FUNCTION_BLOCK List_Person_Test EXTENDS TcUnit.FB_TestSuite

AddAndGet();
AddAndGetShouldBeByReference();
GetCapacity();
GetCount();
Clear();
RemoveAt();
RemoveRange();
Contains();
Exists();
Find();
FindAll();
FindIndex();
FindLast();
FindLastIndex();
Foreach();

METHOD AddAndGet
VAR
    list_Person_ : List_Person_;
    expectedPerson : Person;
    expectedAge : INT := 10;
    expectedIndex : INT := 0;
    actualPtPerson : POINTER TO Person;
    actualAge : INT;
    actualIndex : INT;
END_VAR
TEST('AddAndGetPersonShouldPass');

//Assign
expectedPerson.SetAge(expectedAge);

//Act
actualIndex := list_Person_.AddItem(expectedPerson);
actualPtPerson := list_Person_.GetItem(actualIndex);
actualAge := actualPtPerson^.GetAge();

//Assert
AssertEquals(expectedIndex, actualIndex,'');
AssertEquals(expectedAge, actualAge,'');
AssertTrue(actualPtPerson^.Equals(expectedPerson),'');


TEST_FINISHED();
END_METHOD

METHOD AddAndGetShouldBeByReference
VAR
    list_Person_ : List_Person_;
    expectedPerson : Person;
    expectedAge : INT := 10;
    actualPtPerson : POINTER TO Person;
    actualAge : INT;
END_VAR
TEST('AddAndGetShouldBeByReference');

//Assign

//Act
list_Person_.AddItem(expectedPerson);
actualPtPerson := list_Person_.GetItem(0);
expectedPerson.SetAge(expectedAge);
actualAge := actualPtPerson^.GetAge();

//Assert
AssertEquals(expectedAge, actualAge,'');


TEST_FINISHED();
END_METHOD

METHOD Clear
VAR
    list_Person_ : List_Person_;
    person : Person;
    expectedCount : INT := 1;
    actualCount : INT;
END_VAR
TEST('ClearShouldPass');

//Assign
list_Person_.AddItem(person);

//Act
actualCount := list_Person_.GetCount();

//Assert
AssertEquals(expectedCount, actualCount,'Get count after adding a person');

//Act
list_Person_.Clear();
actualCount := list_Person_.GetCount();

//Assert
expectedCount := 0;
AssertEquals(expectedCount, actualCount,'Get count after clearing the list');


TEST_FINISHED();
END_METHOD

METHOD Contains
VAR
    list_Person_ : List_Person_;
    personA : Person;
    personB : Person;
    personC : Person;
    personD : Person;
    personE : Person;
    personF : Person;
    personG : Person;
    actual : BOOL;
    expected : BOOL := TRUE;
END_VAR
TEST('ContainsShouldPass');

//Assign
personA.SetAge(10);
personB.SetAge(11);
personC.SetAge(12);
personD.SetAge(13);
personE.SetAge(14);
personF.SetAge(15);
personG.SetAge(16);
personA.SetName('A');
personB.SetName('B');
personC.SetName('C');
personD.SetName('D');
personE.SetName('E');
personF.SetName('F');
personG.SetName('G');
list_Person_.AddItem(personA);
list_Person_.AddItem(personB);
list_Person_.AddItem(personC);
list_Person_.AddItem(personD);
list_Person_.AddItem(personE);
list_Person_.AddItem(personF);

//Act
actual := list_Person_.Contains(personC);

//Assert
AssertEquals(expected, actual,'Looking for personC');

//Act
actual := list_Person_.Contains(personG);

//Assert
expected := FALSE;
AssertEquals(expected, actual,'Looking for personG');


TEST_FINISHED();
END_METHOD

METHOD Exists
VAR
    list_Person_ : List_Person_;
    personA : Person;
    personB : Person;
    personC : Person;
    personD : Person;
    personE : Person;
    personF : Person;
    personG : Person;
    predicate_Person_ : Predicate_Person_;
    actual : BOOL;
    expected : BOOL := TRUE;
END_VAR
TEST('ExistsShouldPass');

//Assign
personA.SetAge(10);
personB.SetAge(11);
personC.SetAge(12);
personD.SetAge(13);
personE.SetAge(14);
personF.SetAge(15);
personG.SetAge(16);
personA.SetName('A');
personB.SetName('B');
personC.SetName('C');
personD.SetName('D');
personE.SetName('E');
personF.SetName('F');
personG.SetName('G');
list_Person_.AddItem(personA);
list_Person_.AddItem(personB);
list_Person_.AddItem(personC);
list_Person_.AddItem(personD);
list_Person_.AddItem(personE);
list_Person_.AddItem(personF);

//Act
actual := list_Person_.Exists(predicate_Person_, 2);

//Assert
AssertEquals(expected, actual,'Looking for a person with name C');

//Act
actual := list_Person_.Exists(predicate_Person_, 3);

//Assert
expected := FALSE;
AssertEquals(expected, actual,'Looking for a person with name G');


TEST_FINISHED();
END_METHOD

METHOD Find
VAR
    list_Person_ : List_Person_;
    personA : Person;
    personB : Person;
    personC : Person;
    personD : Person;
    personE : Person;
    personF : Person;
    personG : Person;
    predicate_Person_ : Predicate_Person_;
    actualPtPerson : POINTER TO Person;
    nullPtPerson : POINTER TO person := 0;
END_VAR
TEST('FindShouldPass');

//Assign
personA.SetAge(10);
personB.SetAge(11);
personC.SetAge(12);
personD.SetAge(13);
personE.SetAge(14);
personF.SetAge(15);
personG.SetAge(16);
personA.SetName('A');
personB.SetName('B');
personC.SetName('C');
personD.SetName('D');
personE.SetName('E');
personF.SetName('F');
personG.SetName('G');
list_Person_.AddItem(personA);
list_Person_.AddItem(personB);
list_Person_.AddItem(personC);
list_Person_.AddItem(personD);
list_Person_.AddItem(personE);
list_Person_.AddItem(personF);

//Act
actualPtPerson := list_Person_.Find(predicate_Person_, 2);

//Assert
AssertTrue(actualPtPerson^.Equals(personC),'Get person with name C');

//Act
actualPtPerson := list_Person_.Find(predicate_Person_, 3);

//Assert
AssertEquals(nullPtPerson, actualPtPerson,'Get Zero when looking for person with name G');


TEST_FINISHED();
END_METHOD

METHOD FindAll
VAR
    list_Person_ : List_Person_;
    personA : Person;
    personB : Person;
    personC : Person;
    personD : Person;
    personE : Person;
    personF : Person;
    personG : Person;
    predicate_Person_ : Predicate_Person_;
    actualList_Person_ : list_Person_;
    actualCount : INT;
    expectedCount : INT := 3;
    actualPtPerson0 : POINTER TO Person;
    actualPtPerson1 : POINTER TO Person;
    actualPtPerson2 : POINTER TO Person;
END_VAR
TEST('FindAllShouldPass');

//Assign
personA.SetAge(10);
personB.SetAge(11);
personC.SetAge(12);
personD.SetAge(13);
personE.SetAge(14);
personF.SetAge(15);
personG.SetAge(16);
list_Person_.AddItem(personA);
list_Person_.AddItem(personB);
list_Person_.AddItem(personC);
list_Person_.AddItem(personD);
list_Person_.AddItem(personE);
list_Person_.AddItem(personF);

//Act
actualList_Person_ := list_Person_.FindAll(predicate_Person_, 1); //Get people younger than 13
actualCount := actualList_Person_.GetCount();
actualPtPerson0 := actualList_Person_.GetItem(0);
actualPtPerson1 := actualList_Person_.GetItem(1);
actualPtPerson2 := actualList_Person_.GetItem(2);

//Assert
AssertEquals(expectedCount, actualCount, 'Check new list count');
AssertTrue(actualPtPerson0^.Equals(personA),'First element should personA');
AssertTrue(actualPtPerson1^.Equals(personB),'First element should personB');
AssertTrue(actualPtPerson2^.Equals(personC),'First element should personC');

TEST_FINISHED();
END_METHOD

METHOD FindIndex
VAR
    list_Person_ : List_Person_;
    personA : Person;
    personB : Person;
    personC : Person;
    personD : Person;
    personE : Person;
    personF : Person;
    personG : Person;
    predicate_Person_ : Predicate_Person_;
    actualIndex : INT;
    expectedIndex : INT := 2;
END_VAR
TEST('FindIndexShouldPass');

//Assign
personA.SetAge(10);
personB.SetAge(11);
personC.SetAge(12);
personD.SetAge(13);
personE.SetAge(14);
personF.SetAge(15);
personG.SetAge(16);
personA.SetName('A');
personB.SetName('B');
personC.SetName('C');
personD.SetName('D');
personE.SetName('E');
personF.SetName('F');
personG.SetName('G');
list_Person_.AddItem(personA);
list_Person_.AddItem(personB);
list_Person_.AddItem(personC);
list_Person_.AddItem(personD);
list_Person_.AddItem(personE);
list_Person_.AddItem(personF);

//Act
actualIndex := list_Person_.FindIndex(predicate_Person_, 2);

//Assert
AssertEquals(expectedIndex, actualIndex, 'find person with name C index');

//Act
actualIndex := list_Person_.FindIndex(predicate_Person_, 3);

//Assert
expectedIndex := -1;
AssertEquals(expectedIndex, actualIndex, 'Find person with name G index');


TEST_FINISHED();
END_METHOD

METHOD FindLast
VAR
    list_Person_ : List_Person_;
    personA : Person;
    personB : Person;
    personC : Person;
    personC2 : Person;
    personD : Person;
    personE : Person;
    personF : Person;
    personG : Person;
    predicate_Person_ : Predicate_Person_;
    actualPtPerson : POINTER TO Person;
    nullPtPerson : POINTER TO person := 0;
END_VAR
TEST('FindLastShouldPass');

//Assign
personA.SetAge(10);
personB.SetAge(11);
personC.SetAge(12);
personC2.SetAge(22);
personD.SetAge(13);
personE.SetAge(14);
personF.SetAge(15);
personG.SetAge(16);
personA.SetName('A');
personB.SetName('B');
personC.SetName('C');
personC2.SetName('C');
personD.SetName('D');
personE.SetName('E');
personF.SetName('F');
personG.SetName('G');
list_Person_.AddItem(personA);
list_Person_.AddItem(personB);
list_Person_.AddItem(personC);
list_Person_.AddItem(personD);
list_Person_.AddItem(personE);
list_Person_.AddItem(personC2); //Duplicated C
list_Person_.AddItem(personF);

//Act
actualPtPerson := list_Person_.FindLast(predicate_Person_, 2);

//Assert
AssertFalse(actualPtPerson^.Equals(personC),'Not the last person with name C');
AssertTrue(actualPtPerson^.Equals(personC2),'Be the last person with name C');

//Act
actualPtPerson := list_Person_.Find(predicate_Person_, 3);

//Assert
AssertEquals(nullPtPerson, actualPtPerson,'Get Zero when looking for person with name G');


TEST_FINISHED();
END_METHOD

METHOD FindLastIndex
VAR
    list_Person_ : List_Person_;
    personA : Person;
    personB : Person;
    personC : Person;
    personC2 : Person;
    personD : Person;
    personE : Person;
    personF : Person;
    personG : Person;
    predicate_Person_ : Predicate_Person_;
    actualIndex : INT;
    expectedIndex : INT := 5;
END_VAR
TEST('FindLastIndexShouldPass');

//Assign
personA.SetAge(10);
personB.SetAge(11);
personC.SetAge(12);
personC.SetAge(22);
personD.SetAge(13);
personE.SetAge(14);
personF.SetAge(15);
personG.SetAge(16);
personA.SetName('A');
personB.SetName('B');
personC.SetName('C');
personC2.SetName('C');
personD.SetName('D');
personE.SetName('E');
personF.SetName('F');
personG.SetName('G');
list_Person_.AddItem(personA);
list_Person_.AddItem(personB);
list_Person_.AddItem(personC);
list_Person_.AddItem(personD);
list_Person_.AddItem(personE);
list_Person_.AddItem(personC2);
list_Person_.AddItem(personF);

//Act
actualIndex := list_Person_.FindLastIndex(predicate_Person_, 2);

//Assert
AssertEquals(expectedIndex, actualIndex, 'Find last person with name C index');

//Act
actualIndex := list_Person_.FindLastIndex(predicate_Person_, 3);

//Assert
expectedIndex := -1;
AssertEquals(expectedIndex, actualIndex, 'Find person with name G index');


TEST_FINISHED();
END_METHOD

METHOD Foreach
VAR
    list_Person_ : List_Person_;
    personA : Person;
    personB : Person;
    personC : Person;
    personD : Person;
    personE : Person;
    personF : Person;
    personG : Person;
    action_Person_ : Action_Person_;
    actualPtPersonArray : ARRAY[0..3] OF POINTER TO Person;
    j : INT;
    expectedName : STRING := 'John';
END_VAR
TEST('ForeachShouldPass');

//Assign
personA.SetAge(10);
personB.SetAge(11);
personC.SetAge(12);
personD.SetAge(13);
personE.SetAge(14);
personF.SetAge(15);
personG.SetAge(16);
personA.SetName('A');
personB.SetName('B');
personC.SetName('C');
personD.SetName('D');
personE.SetName('E');
personF.SetName('F');
personG.SetName('G');
list_Person_.AddItem(personA);
list_Person_.AddItem(personB);
list_Person_.AddItem(personC);
list_Person_.AddItem(personD);

//Act
list_Person_.Foreach(action_Person_, 2);
FOR j:=0 TO 3 DO
    actualPtPersonArray[j] := list_Person_.GetItem(j);
END_FOR

//Assert
AssertEquals_STRING(expectedName, actualPtPersonArray[0]^.GetName(),'element 0 shuold be named John');
AssertEquals_STRING(expectedName, actualPtPersonArray[1]^.GetName(),'element 0 shuold be named John');
AssertEquals_STRING(expectedName, actualPtPersonArray[2]^.GetName(),'element 0 shuold be named John');
AssertEquals_STRING(expectedName, actualPtPersonArray[3]^.GetName(),'element 0 shuold be named John');


TEST_FINISHED();
END_METHOD

METHOD GetCapacity
VAR
    list_Person_ : List_Person_;
    person : Person;
    expectedCapacity : INT := GVL.LIST_UPPER_BOUND + 1;
    actualCapacity : INT;
END_VAR
TEST('GetCapacityShouldPass');

//Act
actualCapacity := list_Person_.GetCapacity();

//Assert1
AssertEquals_INT(expectedCapacity, actualCapacity,'Get capacity at the begining');


//Assign
list_Person_.AddItem(person);

//Act
actualCapacity := list_Person_.GetCapacity();

//Assert2
AssertEquals(expectedCapacity, actualCapacity,'Get capacity after adding a person');


TEST_FINISHED();
END_METHOD

METHOD GetCount
VAR
    list_Person_ : List_Person_;
    person : Person;
    expectedCount : INT := 0;
    actualCount : INT;
    actualPtPerson : POINTER TO Person;
END_VAR
TEST('GetCountShouldPass');

//Act
actualCount := list_Person_.GetCount();

//Assert
AssertEquals_INT(expectedCount, actualCount,'Get count at the begining');


//Assign
list_Person_.AddItem(person);

//Act
actualCount := list_Person_.GetCount();

//Assert
expectedCount := 1;
AssertEquals(expectedCount, actualCount,'Get count after adding a person');


TEST_FINISHED();
END_METHOD

METHOD RemoveAt
VAR
    list_Person_ : List_Person_;
    person : Person;
    expectedPtPerson : POINTER TO Person := 0;
    expectedCount : INT := 0;
    actualPtPerson : POINTER TO Person;
    actualCount : INT;
END_VAR
TEST('RemoveAtShouldPass');

//Assign
list_Person_.AddItem(person);

//Act
list_Person_.RemoveAt(0);
actualCount := list_Person_.GetCount();
actualPtPerson := list_Person_.GetItem(0);

//Assert
AssertEquals(expectedCount, actualCount,'');
AssertEquals(expectedPtPerson, actualPtPerson,'');


TEST_FINISHED();
END_METHOD

METHOD RemoveRange
VAR
    list_Person_ : List_Person_;
    person0 : Person;
    person1 : Person;
    person2 : Person;
    person3 : Person;
    person4 : Person;
    person5 : Person;
    person6 : Person;
    expectedPtPerson : POINTER TO Person := 0;
    expectedCount : INT := 7 - 3;
    actualPtPerson1 : POINTER TO Person;
    actualPtPerson2 : POINTER TO Person;
    actualCount : INT;
END_VAR
TEST('RemoveRangeShouldPass');

//Assign
person0.SetAge(10);
person1.SetAge(11);
person2.SetAge(12);
person3.SetAge(13);
person4.SetAge(14);
person5.SetAge(15);
person6.SetAge(16);
list_Person_.AddItem(person0);
list_Person_.AddItem(person1);
list_Person_.AddItem(person2);
list_Person_.AddItem(person3);
list_Person_.AddItem(person4);
list_Person_.AddItem(person5);
list_Person_.AddItem(person6);

//Act
list_Person_.RemoveRange(2,3);
actualCount := list_Person_.GetCount();
actualPtPerson1 := list_Person_.GetItem(1);
actualPtPerson2 := list_Person_.GetItem(2);

//Assert
AssertEquals(expectedCount, actualCount,'');
AssertEquals_INT(person1.GetAge(), actualPtPerson1^.GetAge(),'');
AssertEquals_INT(person5.GetAge(), actualPtPerson2^.GetAge(),'');


TEST_FINISHED();
END_METHOD

END_FUNCTION_BLOCK

(* stored: Version 1.1.0.1, ProductVersion 3.1.4024.6
   POU List_Person_Test: Id {f9270774-45f6-4a3c-bd99-dc3e4865897e}, SpecialFunc None
   Method AddAndGet: Id {25c92982-6de9-488f-9bc0-45793e501629}
   Method AddAndGetShouldBeByReference: Id {d5902a8f-61b3-4da7-91e7-b3e1326fada2}
   Method Clear: Id {9b3dfb6f-1f77-47b8-8a33-f0a2c6ffe4cf}
   Method Contains: Id {bcc8c300-f0ae-4774-b872-f70bc7232e4b}
   Method Exists: Id {2d5869da-5a98-40d2-baa2-7f0ec5c9ca2b}
   Method Find: Id {88eff670-7867-4249-acd8-bd79171fc10a}
   Method FindAll: Id {7425f332-49f9-4c20-88f0-da5e69ea77ac}
   Method FindIndex: Id {4d72a505-eb57-4e55-8564-5f47ecafc6e4}
   Method FindLast: Id {abbb3269-33fc-42ca-8bd9-9cbddf8b0564}
   Method FindLastIndex: Id {2ce0d703-0d51-4a15-b8a5-468a2c4b2f32}
   Method Foreach: Id {c7149333-61bc-45db-a517-2be27202cf0d}
   Method GetCapacity: Id {8ddaab13-7598-4afc-a5e5-0cd2f6d7be65}
   Method GetCount: Id {e9e9e69d-bbf9-467d-a81f-09763039079f}
   Method RemoveAt: Id {1d891a18-a23d-45c2-8d94-b094a5a2c29f}
   Method RemoveRange: Id {d6049325-00aa-4c78-a69d-b2138d02581d} *)
